# EPICS StreamDevice protocol: fug-loc/fugApp/Db/fug.proto
OutTerminator = CR LF;
InTerminator  = LF;

ReadTimeout   = 1000;
WriteTimeout  = 1000;
PollPeriod    = 100;
ReplyTimeout  = 1000;
ExtraInput    = Ignore;

## Commands wrote from Probus V documentation (V2.22)

###
# Reset
##
reset {
    out "=";
}

###
# Power
##
get_status {
    ExtraInput = Ignore;
    out ">BON?";
    in  "BON:%d%*4c";
}

set_status {
    out "F%d";
    @init { get_status };
}

query_on_status{
    out ">DON?"
    in "DON:%d"
}

###
# Current
##
get_current {
    ExtraInput = Ignore;
    out ">S1?";
    in  "%*3c%f";
}

set_current {
    ExtraInput = Ignore;
    out ">S1 %f";
    in "E0";
    @init { get_current };
}

measure_current {
    ExtraInput = Ignore;
    out ">M1?";
    in  "%*3c%f";
}

###
# Voltage
##
get_voltage {
    ExtraInput = Ignore;
    out ">S0?";
    in  "%*3c%f";
}

set_voltage {
    ExtraInput = Ignore;
    out ">S0 %f";
    in "E0";
    @init { get_voltage };
}

measure_voltage {
    ExtraInput = Ignore;
    out ">M0?";
    in  "%*3c%f";
}

###
# Ramp
##
set_ramp_mode {
    out ">S0B %d";
    in "E0"
}

get_ramp_mode {
    out ">S0B?";
    in "S0B:%d%*4c"
}

get_ramp_status {
    out ">S0S?";
    in "S0S:%d%*4c"
}

set_ramp_value {
    out ">S0R %f";
    in "E0"
}

get_ramp_value {
    out ">S0R?";
    in "S0R:%f"
}

###
# Other
##

get_serial_number {
    out "*IDN?";
    in  "%39c";
}

set_actual {
    out ">S0A %f";
    in "E0"
}

get_statusbytes {
    out ">KS?";
    in "KS:%d"
}

query_polarity {
    out ">DX?"
    in "DX:%d"
}

set_polarity{
    out ">BX %d";
    in "E0";
}

query_remote_ctrl {
    out ">DSD?"
    in "DSD:%d"
}
